Universal Robots PolyScope program: manual_teleoperation.urp

Program manual_teleoperation (installation=default directory=../programs createdIn=5.9.1.1031110 lastSavedIn=5.9.1.1031110 robotSerialNumber=20195501059)
Calibrated DH parameters: a=[0, -0.425, -0.3922, 0, 0, 0]; d=[0.1625, 0, 0, 0.1333, 0.0997, 0.0996]; alpha=[1.570796, 0, 0, 1.570796, -1.570796, 0]; deltaTheta=[0, 0, 0, 0, 0, 0]
Robot Program (runOnlyOnce=false)
  URCap Teleop (teleop, Olis Robotics) dataModel(OperatorMessage=Manual teleoperation)
  Halt
